FUNCTION_BLOCK FB_ArithMittel10
VAR_INPUT
	iInputValue	: INT;
END_VAR
VAR_OUTPUT
	iOut		: INT;
END_VAR
VAR
	value 		: ARRAY [0..9] OF INT;
	counter		: INT 	:= 0;
	counter2	: INT	:= 0;
	x			: REAL 	:= 0;
	bInit		: BOOL	:= FALSE;
END_VAR


value[counter]  := iInputValue;

//Initialisierung abgeschlossen
IF counter = 9 THEN
	bInit	:= TRUE;
END_IF

IF bInit THEN
	
	x := 0;

	// Berechnung
	FOR counter2 := 0 TO 9 BY 1 DO
    	x := x + value[counter2];
	END_FOR;
		
	x := x / 10;	//Mitteln
	
	iOut := REAL_TO_INT(x);
	
ELSE
	iOut := 0;
END_IF

counter := (counter + 1) MOD 10;

END_FUNCTION_BLOCK

(* stored: Version 1.1.0.1, ProductVersion 3.1.4024.4
   POU FB_ArithMittel10: Id {bb4fc685-38f4-4b86-8ac7-1dd0c17bd73e}, SpecialFunc None *)
